FUNCTION_BLOCK SKILL_Control (* Skill state machine: Start/Stop/Abort/Reset over OPC UA (owner only, Start only in module Execute) and START/HALT/ABORT from a parent; Idle 0, Running 1, Stopping 2, Succeeded 3, Failed 4, Aborted 5; GO starts the execution (FromUa: with the Start arguments, else with the parent's values) *)
  (* Standard: 61499-2 *)
  (* Version 0.1, 2026-09-28, Project contributors, AAU Smart Production Lab *)
  PACKAGE modlib;
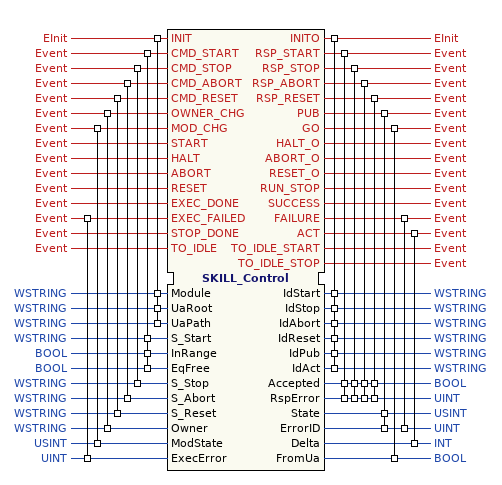
  EVENT_INPUT
    INIT : EInit WITH Module, UaRoot, UaPath;
    CMD_START WITH S_Start, InRange, EqFree;
    CMD_STOP WITH S_Stop;
    CMD_ABORT WITH S_Abort;
    CMD_RESET WITH S_Reset;
    OWNER_CHG WITH Owner;
    MOD_CHG WITH ModState;
    START;
    HALT;
    ABORT;
    RESET;
    EXEC_DONE;
    EXEC_FAILED WITH ExecError;
    STOP_DONE;
    TO_IDLE;
  END_EVENT
  EVENT_OUTPUT
    INITO : EInit WITH IdStart, IdStop, IdAbort, IdReset, IdPub, IdAct;
    RSP_START WITH Accepted, RspError;
    RSP_STOP WITH Accepted, RspError;
    RSP_ABORT WITH Accepted, RspError;
    RSP_RESET WITH Accepted, RspError;
    PUB WITH State, ErrorID;
    GO WITH FromUa;
    HALT_O;
    ABORT_O;
    RESET_O;
    RUN_STOP;
    SUCCESS;
    FAILURE WITH ErrorID;
    ACT WITH Delta;
    TO_IDLE_START;
    TO_IDLE_STOP;
  END_EVENT
  VAR_INPUT
    Module : WSTRING;
    UaRoot : WSTRING;
    UaPath : WSTRING;
    S_Start : WSTRING;
    InRange : BOOL;
    EqFree : BOOL;
    S_Stop : WSTRING;
    S_Abort : WSTRING;
    S_Reset : WSTRING;
    Owner : WSTRING;
    ModState : USINT;
    ExecError : UINT;
  END_VAR
  VAR_OUTPUT
    IdStart : WSTRING;
    IdStop : WSTRING;
    IdAbort : WSTRING;
    IdReset : WSTRING;
    IdPub : WSTRING;
    IdAct : WSTRING;
    Accepted : BOOL;
    RspError : UINT;
    State : USINT;
    ErrorID : UINT;
    Delta : INT;
    FromUa : BOOL;
  END_VAR
  VAR
    Owned : BOOL;
    Here : USINT;
    Active : BOOL;
  END_VAR
  EC_STATES
    START;
    Init : Alg_Init -> INITO;
    Idle : Alg_Idle -> PUB;
    Running : Alg_Running -> PUB;
    Stopping : Alg_Stopping -> PUB;
    StopProc : Alg_StopProc -> PUB;
    Succeeded : Alg_Succeeded -> PUB, -> TO_IDLE_START;
    Failed : Alg_Failed -> PUB;
    Aborted : Alg_Aborted -> PUB;
    GoUa : Alg_GoUa -> ACT, -> TO_IDLE_STOP, -> GO;
    GoParent : Alg_GoParent -> ACT, -> TO_IDLE_STOP, -> GO;
    Halt : -> HALT_O;
    RunStop : -> RUN_STOP;
    Succeed : Alg_Succeed -> ACT, -> SUCCESS;
    Fail : Alg_Fail -> ACT, -> FAILURE;
    Interrupted : Alg_Interrupted -> ACT, -> FAILURE;
    AbortChk;
    AbortActive : Alg_AbortActive -> ABORT_O, -> ACT;
    AbortIdle : -> ABORT_O;
    StartRefused : Alg_StartRefused -> FAILURE;
    ResetOk : -> RESET_O;
    ChkStart : Alg_ChkStart -> RSP_START;
    ChkStop : Alg_ChkStop -> RSP_STOP;
    ChkAbort : Alg_ChkAbort -> RSP_ABORT;
    ChkReset : Alg_ChkReset -> RSP_RESET;
  END_STATES
  EC_TRANSITIONS
    START TO Init := INIT;
    Init TO Idle := 1;
    Idle TO ChkStart := CMD_START;
    Idle TO ChkStop := CMD_STOP;
    Idle TO ChkAbort := CMD_ABORT;
    Idle TO ChkReset := CMD_RESET;
    Running TO ChkStart := CMD_START;
    Running TO ChkStop := CMD_STOP;
    Running TO ChkAbort := CMD_ABORT;
    Running TO ChkReset := CMD_RESET;
    Stopping TO ChkStart := CMD_START;
    Stopping TO ChkStop := CMD_STOP;
    Stopping TO ChkAbort := CMD_ABORT;
    Stopping TO ChkReset := CMD_RESET;
    StopProc TO ChkStart := CMD_START;
    StopProc TO ChkStop := CMD_STOP;
    StopProc TO ChkAbort := CMD_ABORT;
    StopProc TO ChkReset := CMD_RESET;
    Succeeded TO ChkStart := CMD_START;
    Succeeded TO ChkStop := CMD_STOP;
    Succeeded TO ChkAbort := CMD_ABORT;
    Succeeded TO ChkReset := CMD_RESET;
    Failed TO ChkStart := CMD_START;
    Failed TO ChkStop := CMD_STOP;
    Failed TO ChkAbort := CMD_ABORT;
    Failed TO ChkReset := CMD_RESET;
    Aborted TO ChkStart := CMD_START;
    Aborted TO ChkStop := CMD_STOP;
    Aborted TO ChkAbort := CMD_ABORT;
    Aborted TO ChkReset := CMD_RESET;
    Idle TO GoParent := START;
    Succeeded TO GoParent := START;
    Failed TO GoParent := START;
    Aborted TO StartRefused := START;
    StartRefused TO Aborted := 1;
    Running TO Succeed := EXEC_DONE;
    Running TO Fail := EXEC_FAILED;
    Running TO Halt := HALT;
    Running TO Halt := MOD_CHG[(ModState = 7) AND FromUa];
    Stopping TO RunStop := EXEC_DONE;
    Stopping TO RunStop := EXEC_FAILED;
    StopProc TO Interrupted := STOP_DONE;
    Idle TO AbortChk := ABORT;
    Idle TO AbortChk := MOD_CHG[(ModState = 8) OR (ModState = 9)];
    Running TO AbortChk := ABORT;
    Running TO AbortChk := MOD_CHG[(ModState = 8) OR (ModState = 9)];
    Stopping TO AbortChk := ABORT;
    Stopping TO AbortChk := MOD_CHG[(ModState = 8) OR (ModState = 9)];
    StopProc TO AbortChk := ABORT;
    StopProc TO AbortChk := MOD_CHG[(ModState = 8) OR (ModState = 9)];
    Succeeded TO AbortChk := ABORT;
    Succeeded TO AbortChk := MOD_CHG[(ModState = 8) OR (ModState = 9)];
    Failed TO AbortChk := ABORT;
    Failed TO AbortChk := MOD_CHG[(ModState = 8) OR (ModState = 9)];
    Aborted TO ResetOk := MOD_CHG[(ModState = 1) OR (ModState = 2)];
    Aborted TO ResetOk := RESET;
    ResetOk TO Idle := 1;
    GoUa TO Running := 1;
    GoParent TO Running := 1;
    Halt TO Stopping := 1;
    RunStop TO StopProc := 1;
    Succeed TO Succeeded := 1;
    Succeeded TO Idle := TO_IDLE;
    Fail TO Failed := 1;
    Interrupted TO Failed := 1;
    AbortChk TO AbortActive := Active;
    AbortChk TO AbortIdle := 1;
    AbortActive TO Aborted := 1;
    AbortIdle TO Aborted := 1;
    ChkStart TO GoUa := Accepted;
    ChkStart TO Idle := Here = 0;
    ChkStart TO Running := Here = 1;
    ChkStart TO Stopping := Here = 2;
    ChkStart TO StopProc := Here = 3;
    ChkStart TO Succeeded := Here = 4;
    ChkStart TO Failed := Here = 5;
    ChkStart TO Aborted := Here = 6;
    ChkStop TO Halt := Accepted;
    ChkStop TO Idle := Here = 0;
    ChkStop TO Running := Here = 1;
    ChkStop TO Stopping := Here = 2;
    ChkStop TO StopProc := Here = 3;
    ChkStop TO Succeeded := Here = 4;
    ChkStop TO Failed := Here = 5;
    ChkStop TO Aborted := Here = 6;
    ChkAbort TO AbortChk := Accepted;
    ChkAbort TO Idle := Here = 0;
    ChkAbort TO Running := Here = 1;
    ChkAbort TO Stopping := Here = 2;
    ChkAbort TO StopProc := Here = 3;
    ChkAbort TO Succeeded := Here = 4;
    ChkAbort TO Failed := Here = 5;
    ChkAbort TO Aborted := Here = 6;
    ChkReset TO ResetOk := Accepted;
    ChkReset TO Idle := Here = 0;
    ChkReset TO Running := Here = 1;
    ChkReset TO Stopping := Here = 2;
    ChkReset TO StopProc := Here = 3;
    ChkReset TO Succeeded := Here = 4;
    ChkReset TO Failed := Here = 5;
    ChkReset TO Aborted := Here = 6;
  END_TRANSITIONS
  ALGORITHM Alg_Init IN ST:
IdStart := CONCAT(CONCAT(CONCAT("opc_ua[CREATE_METHOD;", CONCAT(UaRoot, UaPath)), "/Start"), "]");
IdStop := CONCAT(CONCAT(CONCAT("opc_ua[CREATE_METHOD;", CONCAT(UaRoot, UaPath)), "/Stop"), "]");
IdAbort := CONCAT(CONCAT(CONCAT("opc_ua[CREATE_METHOD;", CONCAT(UaRoot, UaPath)), "/Abort"), "]");
IdReset := CONCAT(CONCAT(CONCAT("opc_ua[CREATE_METHOD;", CONCAT(UaRoot, UaPath)), "/Reset"), "]");
IdPub := CONCAT(CONCAT(CONCAT(CONCAT(CONCAT("opc_ua[WRITE;", CONCAT(UaRoot, UaPath)), "/State;"), CONCAT(UaRoot, UaPath)), "/ErrorID"), "]");
IdAct := CONCAT(CONCAT("loc[", Module), "/activity]");
  END_ALGORITHM
  ALGORITHM Alg_Idle IN ST:
State := 0;
Here := 0;
  END_ALGORITHM
  ALGORITHM Alg_Running IN ST:
State := 1;
Here := 1;
  END_ALGORITHM
  ALGORITHM Alg_Stopping IN ST:
State := 2;
Here := 2;
  END_ALGORITHM
  ALGORITHM Alg_StopProc IN ST:
State := 2;
Here := 3;
  END_ALGORITHM
  ALGORITHM Alg_Succeeded IN ST:
State := 3;
Here := 4;
  END_ALGORITHM
  ALGORITHM Alg_Failed IN ST:
State := 4;
Here := 5;
  END_ALGORITHM
  ALGORITHM Alg_Aborted IN ST:
State := 5;
Here := 6;
  END_ALGORITHM
  ALGORITHM Alg_GoUa IN ST:
Active := TRUE;
Delta := 1;
ErrorID := 0;
FromUa := TRUE;
  END_ALGORITHM
  ALGORITHM Alg_GoParent IN ST:
Active := TRUE;
Delta := 1;
ErrorID := 0;
FromUa := FALSE;
  END_ALGORITHM
  ALGORITHM Alg_Succeed IN ST:
Active := FALSE;
Delta := -1;
ErrorID := 0;
  END_ALGORITHM
  ALGORITHM Alg_Fail IN ST:
Active := FALSE;
Delta := -1;
ErrorID := ExecError;
  END_ALGORITHM
  ALGORITHM Alg_Interrupted IN ST:
Active := FALSE;
Delta := -1;
ErrorID := 7;
  END_ALGORITHM
  ALGORITHM Alg_AbortActive IN ST:
Active := FALSE;
Delta := -1;
ErrorID := 7;
  END_ALGORITHM
  ALGORITHM Alg_StartRefused IN ST:
ErrorID := 4;
  END_ALGORITHM
  ALGORITHM Alg_ChkStart IN ST:
Owned := (S_Start = Owner) AND (Owner <> "");
Accepted := FALSE;
IF NOT Owned THEN
  RspError := 5;
ELSIF ModState <> 6 THEN
  RspError := 4;
ELSIF (Here = 1) OR (Here = 2) OR (Here = 3) THEN
  RspError := 6;
ELSIF Here = 6 THEN
  RspError := 4;
ELSIF NOT InRange THEN
  RspError := 8;
ELSIF NOT EqFree THEN
  RspError := 6;
ELSE
  Accepted := TRUE;
  RspError := 0;
END_IF;
  END_ALGORITHM
  ALGORITHM Alg_ChkStop IN ST:
Owned := (S_Stop = Owner) AND (Owner <> "");
Accepted := Owned AND (Here = 1);
IF NOT Owned THEN
  RspError := 5;
ELSIF NOT Accepted THEN
  RspError := 4;
ELSE
  RspError := 0;
END_IF;
  END_ALGORITHM
  ALGORITHM Alg_ChkAbort IN ST:
Owned := (S_Abort = Owner) AND (Owner <> "");
Accepted := Owned AND (Here <> 6);
IF NOT Owned THEN
  RspError := 5;
ELSIF NOT Accepted THEN
  RspError := 4;
ELSE
  RspError := 0;
END_IF;
  END_ALGORITHM
  ALGORITHM Alg_ChkReset IN ST:
Owned := (S_Reset = Owner) AND (Owner <> "");
Accepted := Owned AND (Here = 6);
IF NOT Owned THEN
  RspError := 5;
ELSIF NOT Accepted THEN
  RspError := 4;
ELSE
  RspError := 0;
END_IF;
  END_ALGORITHM
END_FUNCTION_BLOCK
